{attribute addProperty BoxType "EL5101-0000-1020"}
{attribute addProperty Id "StatusAT %I*Status_BAA20CF71621Counter_valueAT %I*UINT16217Latch_valueAT %I*UINT16218"}
{attribute addProperty CRC "3942523218"}
{attribute addProperty SizeInBites "48"}
{attribute addProperty SizeInBytes "6"}
TYPE ENC_Status_compact_EAFE2152 :
STRUCT
	{attribute addProperty Name "Status"}
	Status AT %I* : Status_BAA20CF7;
	{attribute addProperty Name "Counter_value"}
	Counter_value AT %I* : UINT;
	{attribute addProperty Name "Latch_value"}
	Latch_value AT %I* : UINT;
END_STRUCT
END_TYPE

(* stored: Version 1.2.0.0, ProductVersion 3.1.4024.9
   DUT ENC_Status_compact_EAFE2152: Id {748a53b8-6180-4c91-a32a-d7aba878d37c} *)
